{attribute addProperty BoxType "EK1122-0000-0018"}
{attribute addProperty Id "Beckhoff_AX86xxsub_EK1100EK1100_179A0949162A_0001_AX8620_0000_0026AX8620_B97EFC7416220.25A_0002_AX8620_0000_0027AX8620_5470AD2416220.25A_0003_AX8620_0000_0029AX8620_4A92314216220.25A_0004_AX8620_0000_0030AX8620_4A92314216220.25A_0005_AX8620_0000_0031AX8620_4A92314216220.25A_0006_AX8620_0000_0032AX8620_4A92314216220.25A_0007_AX8620_0000_0100AX8620_4A92314216220.25A_0008_AX8620_0000_0101AX8620_4A92314216220.25A_0009_AX8620_0000_0102AX8620_4A92314216220.25A_0010_AX8620_0000_0103AX8620_4A92314216220.25A_0011_AX8620_1000_0026AX8620_56141E8A16220.25A_0012_AX8620_1000_0027AX8620_BB1A4FDA16220.25A_0013_AX8620_1000_0029AX8620_4A92314216220.25A_0014_AX8620_1000_0030AX8620_4A92314216220.25A_0015_AX8620_1000_0031AX8620_4A92314216220.25A_0016_AX8620_1000_0032AX8620_4A92314216220.25A_0017_AX8620_1000_0100AX8620_4A92314216220.25A_0018_AX8620_1000_0101AX8620_4A92314216220.25A_0019_AX8640_0000_0026AX8640_56141E8A16220.25A_0020_AX8640_0000_0027AX8640_BB1A4FDA16220.25A_0021_AX8640_0000_0029AX8640_4A92314216220.25A_0022_AX8640_0000_0030AX8640_4A92314216220.25A_0023_AX8640_0000_0031AX8640_4A92314216220.25A_0024_AX8640_0000_0032AX8640_4A92314216220.25A_0025_AX8640_0000_0100AX8640_4A92314216220.25A_0026_AX8640_0000_0101AX8640_4A92314216220.25A_0027_AX8640_0000_0102AX8640_4A92314216220.25A_0028_AX8640_0000_0103AX8640_4A92314216220.25A_0029_AX8640_1000_0026AX8640_56141E8A16220.25A_0030_AX8640_1000_0027AX8640_BB1A4FDA16220.25A_0031_AX8640_1000_0029AX8640_4A92314216220.25A_0032_AX8640_1000_0030AX8640_4A92314216220.25A_0033_AX8640_1000_0031AX8640_4A92314216220.25A_0034_AX8640_1000_0032AX8640_4A92314216220.25A_0035_AX8640_1000_0100AX8640_4A92314216220.25A_0036_AX8640_1000_0101AX8640_4A92314216220.25"}
{attribute addProperty CRC "2657209303"}
{attribute addProperty SizeInBites "5848"}
{attribute addProperty SizeInBytes "731"}
TYPE Beckhoff_AX86xxEK1122_9E61CBD7 EXTENDS EK1122_179A0949 :
STRUCT
	{attribute addProperty Name "Beckhoff_AX86xxsub_EK1100"}
	Beckhoff_AX86xxsub_EK1100 : EK1100_179A0949;
	{attribute addProperty Name "A_0001_AX8620_0000_0026"}
	A_0001_AX8620_0000_0026 : AX8620_B97EFC74;
	{attribute addProperty Name "A_0002_AX8620_0000_0027"}
	A_0002_AX8620_0000_0027 : AX8620_5470AD24;
	{attribute addProperty Name "A_0003_AX8620_0000_0029"}
	A_0003_AX8620_0000_0029 : AX8620_4A923142;
	{attribute addProperty Name "A_0004_AX8620_0000_0030"}
	A_0004_AX8620_0000_0030 : AX8620_4A923142;
	{attribute addProperty Name "A_0005_AX8620_0000_0031"}
	A_0005_AX8620_0000_0031 : AX8620_4A923142;
	{attribute addProperty Name "A_0006_AX8620_0000_0032"}
	A_0006_AX8620_0000_0032 : AX8620_4A923142;
	{attribute addProperty Name "A_0007_AX8620_0000_0100"}
	A_0007_AX8620_0000_0100 : AX8620_4A923142;
	{attribute addProperty Name "A_0008_AX8620_0000_0101"}
	A_0008_AX8620_0000_0101 : AX8620_4A923142;
	{attribute addProperty Name "A_0009_AX8620_0000_0102"}
	A_0009_AX8620_0000_0102 : AX8620_4A923142;
	{attribute addProperty Name "A_0010_AX8620_0000_0103"}
	A_0010_AX8620_0000_0103 : AX8620_4A923142;
	{attribute addProperty Name "A_0011_AX8620_1000_0026"}
	A_0011_AX8620_1000_0026 : AX8620_56141E8A;
	{attribute addProperty Name "A_0012_AX8620_1000_0027"}
	A_0012_AX8620_1000_0027 : AX8620_BB1A4FDA;
	{attribute addProperty Name "A_0013_AX8620_1000_0029"}
	A_0013_AX8620_1000_0029 : AX8620_4A923142;
	{attribute addProperty Name "A_0014_AX8620_1000_0030"}
	A_0014_AX8620_1000_0030 : AX8620_4A923142;
	{attribute addProperty Name "A_0015_AX8620_1000_0031"}
	A_0015_AX8620_1000_0031 : AX8620_4A923142;
	{attribute addProperty Name "A_0016_AX8620_1000_0032"}
	A_0016_AX8620_1000_0032 : AX8620_4A923142;
	{attribute addProperty Name "A_0017_AX8620_1000_0100"}
	A_0017_AX8620_1000_0100 : AX8620_4A923142;
	{attribute addProperty Name "A_0018_AX8620_1000_0101"}
	A_0018_AX8620_1000_0101 : AX8620_4A923142;
	{attribute addProperty Name "A_0019_AX8640_0000_0026"}
	A_0019_AX8640_0000_0026 : AX8640_56141E8A;
	{attribute addProperty Name "A_0020_AX8640_0000_0027"}
	A_0020_AX8640_0000_0027 : AX8640_BB1A4FDA;
	{attribute addProperty Name "A_0021_AX8640_0000_0029"}
	A_0021_AX8640_0000_0029 : AX8640_4A923142;
	{attribute addProperty Name "A_0022_AX8640_0000_0030"}
	A_0022_AX8640_0000_0030 : AX8640_4A923142;
	{attribute addProperty Name "A_0023_AX8640_0000_0031"}
	A_0023_AX8640_0000_0031 : AX8640_4A923142;
	{attribute addProperty Name "A_0024_AX8640_0000_0032"}
	A_0024_AX8640_0000_0032 : AX8640_4A923142;
	{attribute addProperty Name "A_0025_AX8640_0000_0100"}
	A_0025_AX8640_0000_0100 : AX8640_4A923142;
	{attribute addProperty Name "A_0026_AX8640_0000_0101"}
	A_0026_AX8640_0000_0101 : AX8640_4A923142;
	{attribute addProperty Name "A_0027_AX8640_0000_0102"}
	A_0027_AX8640_0000_0102 : AX8640_4A923142;
	{attribute addProperty Name "A_0028_AX8640_0000_0103"}
	A_0028_AX8640_0000_0103 : AX8640_4A923142;
	{attribute addProperty Name "A_0029_AX8640_1000_0026"}
	A_0029_AX8640_1000_0026 : AX8640_56141E8A;
	{attribute addProperty Name "A_0030_AX8640_1000_0027"}
	A_0030_AX8640_1000_0027 : AX8640_BB1A4FDA;
	{attribute addProperty Name "A_0031_AX8640_1000_0029"}
	A_0031_AX8640_1000_0029 : AX8640_4A923142;
	{attribute addProperty Name "A_0032_AX8640_1000_0030"}
	A_0032_AX8640_1000_0030 : AX8640_4A923142;
	{attribute addProperty Name "A_0033_AX8640_1000_0031"}
	A_0033_AX8640_1000_0031 : AX8640_4A923142;
	{attribute addProperty Name "A_0034_AX8640_1000_0032"}
	A_0034_AX8640_1000_0032 : AX8640_4A923142;
	{attribute addProperty Name "A_0035_AX8640_1000_0100"}
	A_0035_AX8640_1000_0100 : AX8640_4A923142;
	{attribute addProperty Name "A_0036_AX8640_1000_0101"}
	A_0036_AX8640_1000_0101 : AX8640_4A923142;
END_STRUCT
END_TYPE

(* stored: Version 1.2.0.0, ProductVersion 3.1.4024.9
   DUT Beckhoff_AX86xxEK1122_9E61CBD7: Id {de962be3-d8a6-4a42-af5f-f3f9431acf5d} *)
